{attribute 'linkalways'} 
{attribute 'no_explicit_call' := 'This FB is a CLASS and must be accessed using methods or properties'}
{attribute 'enable_dynamic_creation'}
FUNCTION_BLOCK FINAL NE_SINT EXTENDS Node
VAR
	in1 : _SINT(0);
	in2 : _SINT(0);
	out : _BOOL(FALSE);
END_VAR

METHOD PUBLIC Clone : I_Node
VAR
	pNode : POINTER TO NE_SINT;
END_VAR
pNode := __NEW(NE_SINT);
Clone := pNode^;
END_METHOD

METHOD FB_init : BOOL
VAR_INPUT
	bInitRetains : BOOL; // if TRUE, the retain variables are initialized (warm start / cold start)
	bInCopyCode : BOOL;  // if TRUE, the instance afterwards gets moved into the copy code (online change)
END_VAR
AddInput('in1',THIS^.in1);
AddInput('in2',THIS^.in2);
AddOutput('out', THIS^.out);
END_METHOD

METHOD PROTECTED OnExecute
VAR
END_VAR
out.Value := in1.Value <> in2.Value;
END_METHOD

END_FUNCTION_BLOCK

(* stored: Version 1.1.0.1, ProductVersion 3.1.4024.15
   POU NE_SINT: Id {d8695d9e-e2ae-4716-b35d-d633ad59a6cf}, SpecialFunc None
   Folder Constructor: Id {3848ddcb-3a5b-443d-b5ab-51a6325183cb}
   Method Clone: Id {31b94ceb-b80e-4ba0-bc56-849e7ae549cf}
   Method FB_init: Id {acffa3e3-7a19-43f4-9478-799c3addb422}
   Method OnExecute: Id {fe380fbf-1b01-468f-978e-015818147130} *)
